// TIA Portal V16 export
// export: Created 2023-09-11T12:14:55.0236389Z, ExportSetting WithDefaults, DisplayName Totally Integrated Automation Portal, DisplayVersion V16 Update 6, DisplayName TIA Portal Version Control Interface, DisplayVersion V16 Update 2, DisplayName TIA Portal Openness, DisplayVersion V16 Update 6, DisplayName STEP 7 Professional, DisplayVersion V16 Update 6, DisplayName STEP 7 Safety, DisplayVersion V16, DisplayName WinCC Advanced, DisplayVersion V16 Update 6
FUNCTION "06_M_Control mode control" : Void   // FC27, LAD
{ S7_Optimized_Access := 'TRUE' }
AUTHOR : rtecmer
VERSION : 0.1
// Kontrola trybu pracy Manual/Automat. Kontrola trybu pracy PID tryb 4 / tryb 3. Sprawdzanie stanu otwarcia Z11, Z12. Sprawdzanie sygnału Alarm Suchobieg. Tryb sterownia zostaje przerwany w wypadku wystąpienia 'Suchobiegu", lub zamknięcia obu zasów Z11 i Z12
// stored: AutoNumber true, IsIECCheckEnabled false, SetENOAutomatically false, UDAEnableTagReadback false
   VAR_IN_OUT
      Timer_Reset_delay : TOF_TIME;
   END_VAR
   VAR_TEMP   // added for the SCL form of the ladder/FBD networks
      _w1 : Bool;
      _w2 : Bool;
   END_VAR
BEGIN

REGION Network 2: bit sygnalizacji pracy w automacie zestawu
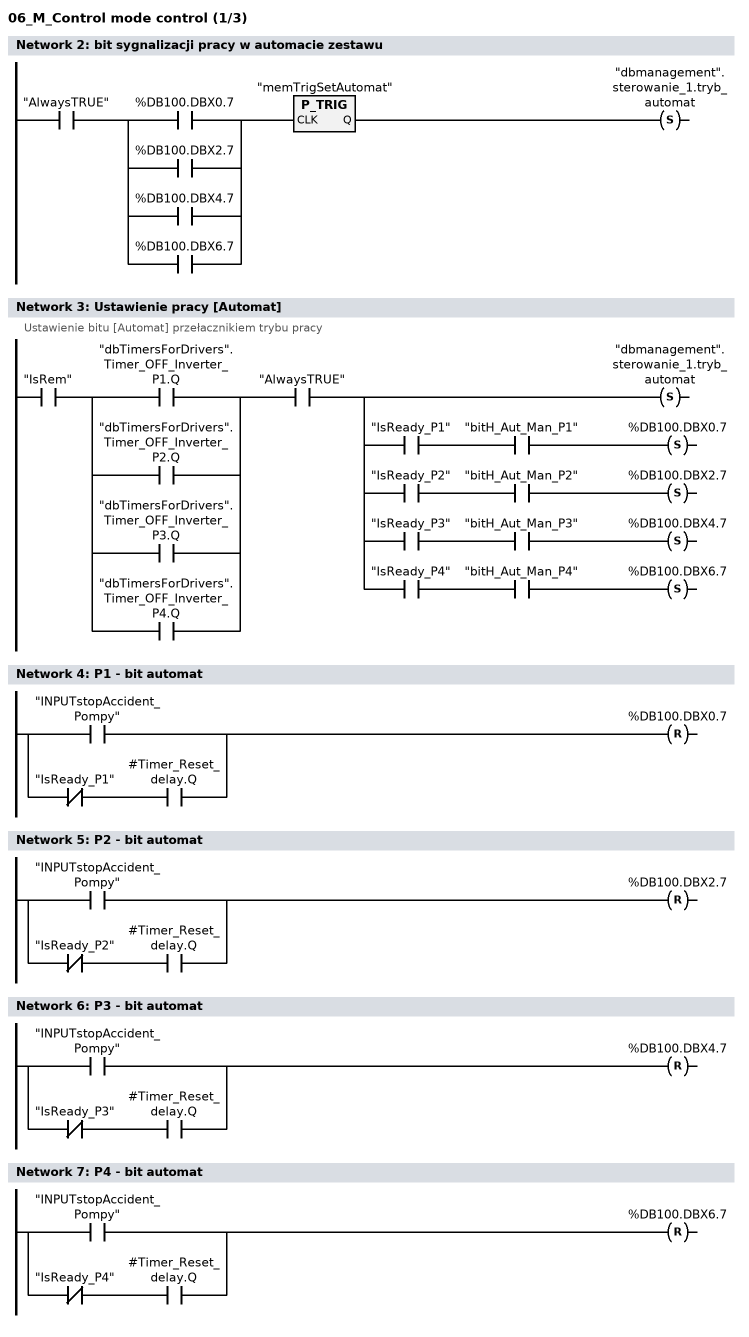
   RUNG wire#powerrail
      Contact( "AlwaysTRUE" )
      wire#w1
      Contact( %DB100.DBX0.7 )
      wire#w2
      P_Trig( "memTrigSetAutomat" )
      S_Coil( "dbmanagement".sterowanie_1.tryb_automat )
   END_RUNG
   RUNG wire#w1
      Contact( %DB100.DBX2.7 )
   END_RUNG wire#w2
   RUNG wire#w1
      Contact( %DB100.DBX4.7 )
   END_RUNG wire#w2
   RUNG wire#w1
      Contact( %DB100.DBX6.7 )
   END_RUNG wire#w2
   // the same network as SCL:
   #_w1 := "AlwaysTRUE" AND (%DB100.DBX0.7 OR %DB100.DBX2.7 OR %DB100.DBX4.7 OR %DB100.DBX6.7);
   #_w2 := #_w1 AND NOT "memTrigSetAutomat";   // rising edge
   "memTrigSetAutomat" := #_w1;
   IF #_w2 THEN "dbmanagement".sterowanie_1.tryb_automat := TRUE; END_IF;
END_REGION

REGION Network 3: Ustawienie pracy [Automat]
   // Ustawienie bitu [Automat] przełacznikiem trybu pracy
   RUNG wire#powerrail
      Contact( "IsRem" )
      wire#w1
      Contact( "dbTimersForDrivers".Timer_OFF_Inverter_P1.Q )
      wire#w2
      Contact( "AlwaysTRUE" )
      wire#w3
      S_Coil( "dbmanagement".sterowanie_1.tryb_automat )
   END_RUNG
   RUNG wire#w1
      Contact( "dbTimersForDrivers".Timer_OFF_Inverter_P2.Q )
   END_RUNG wire#w2
   RUNG wire#w1
      Contact( "dbTimersForDrivers".Timer_OFF_Inverter_P3.Q )
   END_RUNG wire#w2
   RUNG wire#w1
      Contact( "dbTimersForDrivers".Timer_OFF_Inverter_P4.Q )
   END_RUNG wire#w2
   RUNG wire#w3
      Contact( "IsReady_P1" )
      Contact( "bitH_Aut_Man_P1" )
      S_Coil( %DB100.DBX0.7 )
   END_RUNG
   RUNG wire#w3
      Contact( "IsReady_P2" )
      Contact( "bitH_Aut_Man_P2" )
      S_Coil( %DB100.DBX2.7 )
   END_RUNG
   RUNG wire#w3
      Contact( "IsReady_P3" )
      Contact( "bitH_Aut_Man_P3" )
      S_Coil( %DB100.DBX4.7 )
   END_RUNG
   RUNG wire#w3
      Contact( "IsReady_P4" )
      Contact( "bitH_Aut_Man_P4" )
      S_Coil( %DB100.DBX6.7 )
   END_RUNG
   // the same network as SCL:
   #_w1 := "IsRem" AND ("dbTimersForDrivers".Timer_OFF_Inverter_P1.Q OR "dbTimersForDrivers".Timer_OFF_Inverter_P2.Q OR "dbTimersForDrivers".Timer_OFF_Inverter_P3.Q OR "dbTimersForDrivers".Timer_OFF_Inverter_P4.Q) AND "AlwaysTRUE";
   IF #_w1 THEN "dbmanagement".sterowanie_1.tryb_automat := TRUE; END_IF;
   IF #_w1 AND "IsReady_P1" AND "bitH_Aut_Man_P1" THEN %DB100.DBX0.7 := TRUE; END_IF;
   IF #_w1 AND "IsReady_P2" AND "bitH_Aut_Man_P2" THEN %DB100.DBX2.7 := TRUE; END_IF;
   IF #_w1 AND "IsReady_P3" AND "bitH_Aut_Man_P3" THEN %DB100.DBX4.7 := TRUE; END_IF;
   IF #_w1 AND "IsReady_P4" AND "bitH_Aut_Man_P4" THEN %DB100.DBX6.7 := TRUE; END_IF;
END_REGION

REGION Network 4: P1 - bit automat
   RUNG wire#powerrail
      Contact( "INPUTstopAccident_Pompy" )
      wire#w1
      R_Coil( %DB100.DBX0.7 )
   END_RUNG
   RUNG wire#powerrail
      I_Contact( "IsReady_P1" )
      Contact( #Timer_Reset_delay.Q )
   END_RUNG wire#w1
   // the same network as SCL:
   IF "INPUTstopAccident_Pompy" OR (NOT "IsReady_P1" AND #Timer_Reset_delay.Q) THEN
       %DB100.DBX0.7 := FALSE;
   END_IF;
END_REGION

REGION Network 5: P2 - bit automat
   RUNG wire#powerrail
      Contact( "INPUTstopAccident_Pompy" )
      wire#w1
      R_Coil( %DB100.DBX2.7 )
   END_RUNG
   RUNG wire#powerrail
      I_Contact( "IsReady_P2" )
      Contact( #Timer_Reset_delay.Q )
   END_RUNG wire#w1
   // the same network as SCL:
   IF "INPUTstopAccident_Pompy" OR (NOT "IsReady_P2" AND #Timer_Reset_delay.Q) THEN
       %DB100.DBX2.7 := FALSE;
   END_IF;
END_REGION

REGION Network 6: P3 - bit automat
   RUNG wire#powerrail
      Contact( "INPUTstopAccident_Pompy" )
      wire#w1
      R_Coil( %DB100.DBX4.7 )
   END_RUNG
   RUNG wire#powerrail
      I_Contact( "IsReady_P3" )
      Contact( #Timer_Reset_delay.Q )
   END_RUNG wire#w1
   // the same network as SCL:
   IF "INPUTstopAccident_Pompy" OR (NOT "IsReady_P3" AND #Timer_Reset_delay.Q) THEN
       %DB100.DBX4.7 := FALSE;
   END_IF;
END_REGION

REGION Network 7: P4 - bit automat
   RUNG wire#powerrail
      Contact( "INPUTstopAccident_Pompy" )
      wire#w1
      R_Coil( %DB100.DBX6.7 )
   END_RUNG
   RUNG wire#powerrail
      I_Contact( "IsReady_P4" )
      Contact( #Timer_Reset_delay.Q )
   END_RUNG wire#w1
   // the same network as SCL:
   IF "INPUTstopAccident_Pompy" OR (NOT "IsReady_P4" AND #Timer_Reset_delay.Q) THEN
       %DB100.DBX6.7 := FALSE;
   END_IF;
END_REGION

REGION Network 8: bit sygnalizacji pracy w automacie zestawu
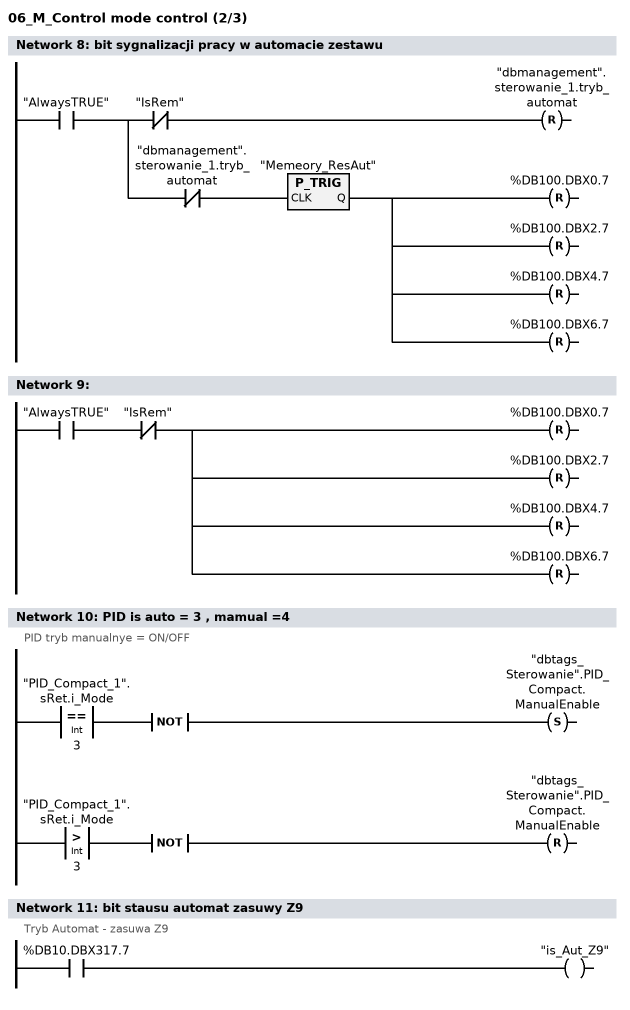
   RUNG wire#powerrail
      Contact( "AlwaysTRUE" )
      wire#w1
      I_Contact( "IsRem" )
      R_Coil( "dbmanagement".sterowanie_1.tryb_automat )
   END_RUNG
   RUNG wire#w1
      I_Contact( "dbmanagement".sterowanie_1.tryb_automat )
      P_Trig( "Memeory_ResAut" )
      wire#w2
      R_Coil( %DB100.DBX0.7 )
   END_RUNG
   RUNG wire#w2
      R_Coil( %DB100.DBX2.7 )
   END_RUNG
   RUNG wire#w2
      R_Coil( %DB100.DBX4.7 )
   END_RUNG
   RUNG wire#w2
      R_Coil( %DB100.DBX6.7 )
   END_RUNG
   // the same network as SCL:
   IF "AlwaysTRUE" AND NOT "IsRem" THEN "dbmanagement".sterowanie_1.tryb_automat := FALSE; END_IF;
   #_w1 := "AlwaysTRUE" AND NOT "dbmanagement".sterowanie_1.tryb_automat;
   #_w2 := #_w1 AND NOT "Memeory_ResAut";   // rising edge
   "Memeory_ResAut" := #_w1;
   IF #_w2 THEN
       %DB100.DBX0.7 := FALSE;
       %DB100.DBX2.7 := FALSE;
       %DB100.DBX4.7 := FALSE;
       %DB100.DBX6.7 := FALSE;
   END_IF;
END_REGION

REGION Network 9
   RUNG wire#powerrail
      Contact( "AlwaysTRUE" )
      I_Contact( "IsRem" )
      wire#w1
      R_Coil( %DB100.DBX0.7 )
   END_RUNG
   RUNG wire#w1
      R_Coil( %DB100.DBX2.7 )
   END_RUNG
   RUNG wire#w1
      R_Coil( %DB100.DBX4.7 )
   END_RUNG
   RUNG wire#w1
      R_Coil( %DB100.DBX6.7 )
   END_RUNG
   // the same network as SCL:
   IF "AlwaysTRUE" AND NOT "IsRem" THEN
       %DB100.DBX0.7 := FALSE;
       %DB100.DBX2.7 := FALSE;
       %DB100.DBX4.7 := FALSE;
       %DB100.DBX6.7 := FALSE;
   END_IF;
END_REGION

REGION Network 10: PID is auto = 3 , mamual =4
   // PID tryb manualnye = ON/OFF
   RUNG wire#powerrail
      { S7_Templates := "SrcType := Int" } EQ_Contact(in1 := "PID_Compact_1".sRet.i_Mode, in2 := 3)
      Not()
      S_Coil( "dbtags_Sterowanie".PID_Compact.ManualEnable )
   END_RUNG
   RUNG wire#powerrail
      { S7_Templates := "SrcType := Int" } GT_Contact(in1 := "PID_Compact_1".sRet.i_Mode, in2 := 3)
      Not()
      R_Coil( "dbtags_Sterowanie".PID_Compact.ManualEnable )
   END_RUNG
   // the same network as SCL:
   IF NOT ("PID_Compact_1".sRet.i_Mode = 3) THEN
       "dbtags_Sterowanie".PID_Compact.ManualEnable := TRUE;
   END_IF;
   IF NOT ("PID_Compact_1".sRet.i_Mode > 3) THEN
       "dbtags_Sterowanie".PID_Compact.ManualEnable := FALSE;
   END_IF;
END_REGION

REGION Network 11: bit stausu automat zasuwy Z9
   // Tryb Automat - zasuwa Z9
   RUNG wire#powerrail
      Contact( %DB10.DBX317.7 )
      Coil( "is_Aut_Z9" )
   END_RUNG
   // the same network as SCL:
   "is_Aut_Z9" := %DB10.DBX317.7;
END_REGION

REGION Network 12: ustawienie bitu automat tryb pracy P1-P4
   // Jeśli REM = 1 i IsModeAut =1  to załącz PID na wartość zadaną
   // Jeśli REM = 0 to reset PID i ustaw tryb 0 (nieaktywny)
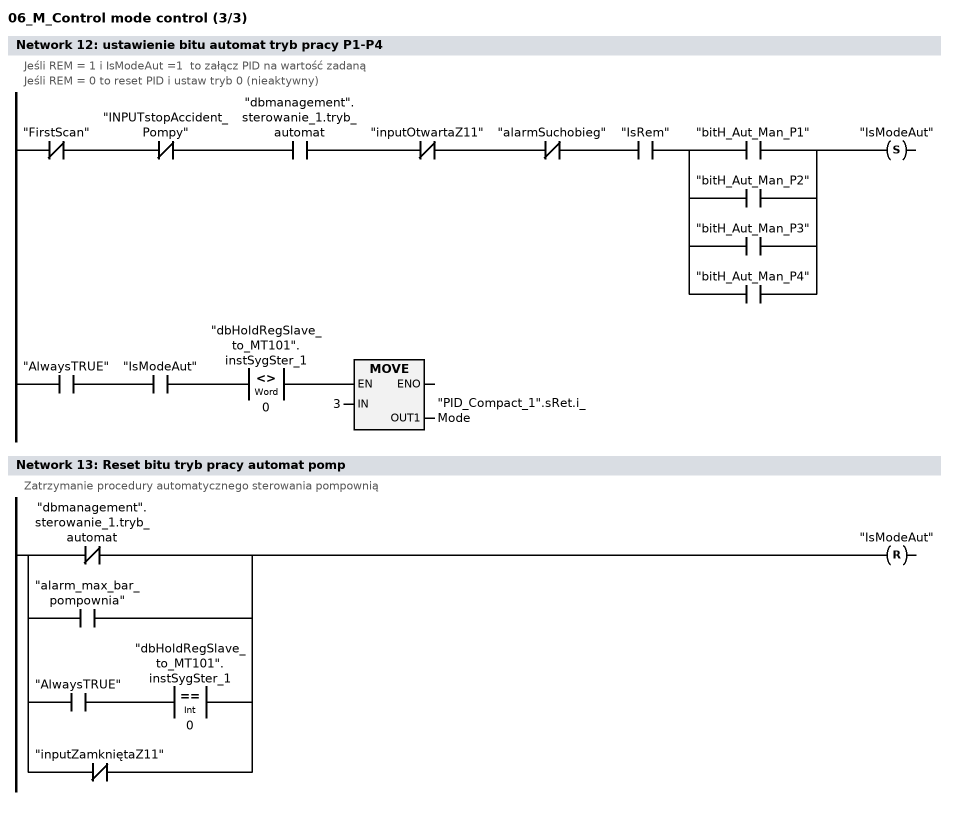
   RUNG wire#powerrail
      I_Contact( "FirstScan" )
      I_Contact( "INPUTstopAccident_Pompy" )
      Contact( "dbmanagement".sterowanie_1.tryb_automat )
      I_Contact( "inputOtwartaZ11" )
      I_Contact( "alarmSuchobieg" )
      Contact( "IsRem" )
      wire#w1
      Contact( "bitH_Aut_Man_P1" )
      wire#w2
      S_Coil( "IsModeAut" )
   END_RUNG
   RUNG wire#w1
      Contact( "bitH_Aut_Man_P2" )
   END_RUNG wire#w2
   RUNG wire#w1
      Contact( "bitH_Aut_Man_P3" )
   END_RUNG wire#w2
   RUNG wire#w1
      Contact( "bitH_Aut_Man_P4" )
   END_RUNG wire#w2
   RUNG wire#powerrail
      Contact( "AlwaysTRUE" )
      Contact( "IsModeAut" )
      { S7_Templates := "SrcType := Word" } NE_Contact(in1 := "dbHoldRegSlave_to_MT101".instSygSter_1, in2 := 0)
      { S7_GenerateENO := "TRUE" } Move(in := 3, out1 => "PID_Compact_1".sRet.i_Mode)
   END_RUNG
   // the same network as SCL:
   IF NOT "FirstScan" AND NOT "INPUTstopAccident_Pompy" AND "dbmanagement".sterowanie_1.tryb_automat AND NOT "inputOtwartaZ11" AND NOT "alarmSuchobieg" AND "IsRem" AND ("bitH_Aut_Man_P1" OR "bitH_Aut_Man_P2" OR "bitH_Aut_Man_P3" OR "bitH_Aut_Man_P4") THEN
       "IsModeAut" := TRUE;
   END_IF;
   IF "AlwaysTRUE" AND "IsModeAut" AND ("dbHoldRegSlave_to_MT101".instSygSter_1 <> 0) THEN
       "PID_Compact_1".sRet.i_Mode := 3;
   END_IF;
END_REGION

REGION Network 13: Reset bitu tryb pracy automat pomp
   // Zatrzymanie procedury automatycznego sterowania pompownią
   RUNG wire#powerrail
      I_Contact( "dbmanagement".sterowanie_1.tryb_automat )
      wire#w1
      R_Coil( "IsModeAut" )
   END_RUNG
   RUNG wire#powerrail
      Contact( "alarm_max_bar_pompownia" )
   END_RUNG wire#w1
   RUNG wire#powerrail
      Contact( "AlwaysTRUE" )
      { S7_Templates := "SrcType := Int" } EQ_Contact(in1 := "dbHoldRegSlave_to_MT101".instSygSter_1, in2 := 0)
   END_RUNG wire#w1
   RUNG wire#powerrail
      I_Contact( "inputZamkniętaZ11" )
   END_RUNG wire#w1
   // the same network as SCL:
   IF NOT "dbmanagement".sterowanie_1.tryb_automat OR "alarm_max_bar_pompownia" OR ("AlwaysTRUE" AND ("dbHoldRegSlave_to_MT101".instSygSter_1 = 0)) OR NOT "inputZamkniętaZ11" THEN
       "IsModeAut" := FALSE;
   END_IF;
END_REGION
END_FUNCTION
